(* IEC 61131-3 sources: rustmatic/structured-text/tests/data, 7 files *)

(* ---- function_block.st ---- *)
FUNCTION_BLOCK FB_Timed_Counter
    //=======================================================================
    // Function Block Timed Counter :  Incremental count of the timed interval
    //=======================================================================
    VAR_INPUT
        Execute         : BOOL := FALSE;        // Trigger signal to begin Timed Counting
        Time_Increment  : REAL := 1.25;         // Enter Cycle Time (Seconds) between counts
        Count_Cycles    : INT  := 20;           // Number of Desired Count Cycles
    END_VAR

    VAR_OUTPUT
        Timer_Done_Bit  : BOOL := FALSE;        // One Shot Bit indicating Timer Cycle Done
        Count_Complete  : BOOL := FALSE;        // Output Bit indicating the Count is complete
        Current_Count   : INT  := 0;            // Accumulating Value of Counter
    END_VAR

    VAR
        CycleTimer      : TON;                  // Timer FB from Command Library
        CycleCounter    : CTU;                  // Counter FB from Command Library
        TimerPreset     : TIME;                 // Converted Time_Increment in Seconds to MS
    END_VAR

    // Start of Function Block programming
    TimerPreset := REAL_TO_TIME(in := Time_Increment) * 1000;

    CycleTimer(
        in := Execute AND NOT CycleTimer.Q,
        pt := TimerPreset);

    Timer_Done_Bit := CycleTimer.Q;

    CycleCounter(
        cu := CycleTimer.Q,
        r := NOT Execute,
        pv := Count_Cycles);

    Current_Count := CycleCounter.cv;
    Count_Complete := CycleCounter.q;

END_FUNCTION_BLOCK

// https://en.wikipedia.org/wiki/Structured_text#Function_block_example

(* ---- case_statement.st ---- *)
CASE i OF
    0:
        i:=1;
    1:
        i:=2;
    2:
        i:=3;
    3:
        i:=0;
    ELSE
        i := -1;
END_CASE

(* ---- first_wikipedia_sample.st ---- *)
// See https://en.wikipedia.org/wiki/Structured_text#Additional_ST_programming_examples
// PLC configuration
CONFIGURATION DefaultCfg
    VAR_GLOBAL
        b_Start_Stop  : BOOL;         // Global variable to represent a boolean.
        b_ON_OFF      : BOOL;         // Global variable to represent a boolean.
        Start_Stop AT %IX0.0:BOOL;    // Digital   input of the PLC (Address 0.0)
        ON_OFF     AT %QX0.0:BOOL;    // Digital output of the PLC (Address 0.0). (Coil)
    END_VAR

    // Schedule the main program to be executed every 20 ms
    TASK Tick(INTERVAL := t#20ms);

    PROGRAM Main WITH Tick : Monitor_Start_Stop;
END_CONFIGURATION

PROGRAM Monitor_Start_Stop          // Actual Program
    VAR_EXTERNAL
        Start_Stop  : BOOL;
        ON_OFF      : BOOL;
    END_VAR
    VAR                             // Temporary variables for logic handling
        ONS_Trig    : BOOL;
        Rising_ONS  : BOOL;
    END_VAR

    // Start of Logic
    // Catch the Rising Edge One Shot of the Start_Stop input
    ONS_Trig    := Start_Stop AND NOT Rising_ONS;

    // Main Logic for Run_Contact -- Toggle ON / Toggle OFF ---
    ON_OFF := (ONS_Trig AND NOT ON_OFF) OR (ON_OFF AND NOT ONS_Trig);

    // Rising One Shot logic
    Rising_ONS := Start_Stop;
END_PROGRAM

(* ---- function_and_program.st ---- *)
PROGRAM stexample
  VAR
    x : BOOL;
  END_VAR
  x := TRUE;
  REPEAT
    x := FALSE;
  UNTIL x := FALSE;
  END_REPEAT;
END_PROGRAM;

FUNCTION add: INT
    VAR_INPUT
        a: INT;
        b: INT;
    END_VAR
    VAR_OUTPUT
        result: INT;
    END_VAR

    result := a + b;
END_FUNCTION;

(* ---- if_chain.st ---- *)
IF S1 = 0 THEN
    S1:= S1+1;
ELSIF S1 = 1 THEN
    S1:= 2;
ELSIF S1 = 2 THEN
    S1:= 3;
ELSE
    S1:=4;
END_IF

// https://owlcation.com/stem/Introduction-to-Structured-Text-With-Codesys-35#mod_46205970

(* ---- if_start_while_initialized_prime_system.st ---- *)
// https://owlcation.com/stem/Introduction-to-Structured-Text-With-Codesys-35#mod_46205880
IF Start THEN
    Start:=FALSE; //Remove Start Latch
    WHILE Initialised = FALSE DO
        System_Prime:=TRUE; //Set Output On For System Primer
    END_WHILE
    System_Prime:=FALSE; //Turn Off Output For System Primer Once Initialised
END_IF

(* ---- simple_program.st ---- *)
PROGRAM stexample
  VAR
    x : BOOL;
  END_VAR
  x := TRUE;
  REPEAT
    x := FALSE;
  UNTIL x := FALSE;
  END_REPEAT;
END_PROGRAM;

// https://www.plcacademy.com/structured-text-tutorial/
